// TIA Portal V19 export
DATA_BLOCK "OT Comms DB"   // DB50
VERSION : 0.0
// stored: AutoNumber false, InstanceOfName OT Comms, InstanceOfType FB
"OT Comms"
   // VAR
   //    get_AlcipM3 : GET;
   //    put_AlcipM3 : PUT;
   //    get_FP_Alsafe : GET;
   //    put_FP_Alsafe : PUT;
   //    FM_PutReq : Bool;
   //    FP_PutReq : Bool;
   //    PutReq : Bool;
   //    PutDone : Bool;
   //    PutError : Bool;
   //    PutMaxTime : Bool;
   //    PutStatus : Word;
   //    FM_GetReq : Bool;
   //    FP_GetReq : Bool;
   //    GetReq : Bool;
   //    GetDone : Bool;
   //    GetError : Bool;
   //    GetMaxTime : Bool;
   //    GetWDFault : Bool;
   //    GetStatus : Word;
   //    FM_GetReq_1 : Bool;
   //    FP_GetReq_1 : Bool;
   //    GetReq_1 : Bool;
   //    GetDone_1 : Bool;
   //    GetError_1 : Bool;
   //    GetMaxTime_1 : Bool;
   //    GetWDFault_1 : Bool;
   //    GetStatus_1 : Word;
   //    GetWatchdog_1 : Int;
   //    FM_PutReq_1 : Bool;
   //    FP_PutReq_1 : Bool;
   //    GetReq_2 : Bool;
   //    GetWatchdog : Int;
   //    PutReq_1 : Bool;
   //    PutDone_1 : Bool;
   //    PutError_1 : Bool;
   //    PutMaxTime_1 : Bool;
   //    PutStatus_1 : Word;
   //    count : Int;
   //    fpCnt : Bool;
   //    ActConnection1 : Bool;
   //    ActConnection2 : Bool;
   //    id : Word;
   //    srcDB : Int;
   //    srcByte : Int;
   //    srcType : Bool;
   //    srcLen : Int;
   //    desDB : Int;
   //    desByte : Int;
   //    desType : Bool;
   //    DesLen : Int;
   // END_VAR
BEGIN
END_DATA_BLOCK
